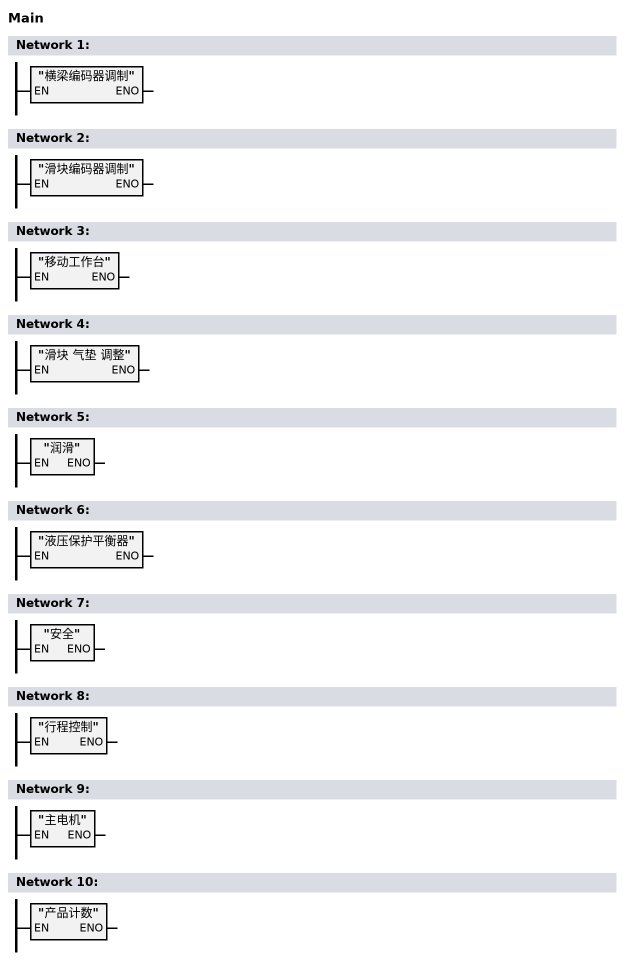
   RUNG wire#powerrail
      "横梁编码器调制"()
   END_RUNG
   // the same network as SCL:
   "横梁编码器调制"();
END_REGION

REGION Network 2
   RUNG wire#powerrail
      "滑块编码器调制"()
   END_RUNG
   // the same network as SCL:
   "滑块编码器调制"();
END_REGION

REGION Network 3
   RUNG wire#powerrail
      "移动工作台"()
   END_RUNG
   // the same network as SCL:
   "移动工作台"();
END_REGION

REGION Network 4
   RUNG wire#powerrail
      "滑块 气垫 调整"()
   END_RUNG
   // the same network as SCL:
   "滑块 气垫 调整"();
END_REGION

REGION Network 5
   RUNG wire#powerrail
      "润滑"()
   END_RUNG
   // the same network as SCL:
   "润滑"();
END_REGION

REGION Network 6
   RUNG wire#powerrail
      "液压保护平衡器"()
   END_RUNG
   // the same network as SCL:
   "液压保护平衡器"();
END_REGION

REGION Network 7
   RUNG wire#powerrail
      "安全"()
   END_RUNG
   // the same network as SCL:
   "安全"();
END_REGION

REGION Network 8
   RUNG wire#powerrail
      "行程控制"()
   END_RUNG
   // the same network as SCL:
   "行程控制"();
END_REGION

REGION Network 9
   RUNG wire#powerrail
      "主电机"()
   END_RUNG
   // the same network as SCL:
   "主电机"();
END_REGION

REGION Network 10
   RUNG wire#powerrail
      "产品计数"()
   END_RUNG
   // the same network as SCL:
   "产品计数"();
END_REGION
END_ORGANIZATION_BLOCK

(* ===== HMI "HMI_RT_1" =====
system functions are stored by id; their names below are inferred from use
connection "HMI_连接_1": ETHERNET, S7_1200_OMS

HMI tags "默认变量表"
   "360" : Bool = PLC 360 AT %M204.3, 100 ms
   "10度" : Bool = PLC 10度 AT %M200.0, 100 ms
   "20度" : Bool = PLC 20度 AT %M200.1, 100 ms
   "30度" : Bool = PLC 30度 AT %M200.2, 100 ms
   "40度" : Bool = PLC 40度 AT %M200.3, 100 ms
   "50" : Bool = PLC 50 AT %M200.4, 100 ms
   "60" : Bool = PLC 60 AT %M200.5, 100 ms
   "70" : Bool = PLC 70 AT %M200.6, 100 ms
   "80" : Bool = PLC 80 AT %M200.7, 100 ms
   "90" : Bool = PLC 90 AT %M201.0, 100 ms
   "100" : Bool = PLC 100 AT %M201.1, 100 ms
   "110" : Bool = PLC 110 AT %M201.2, 100 ms
   "120" : Bool = PLC 120 AT %M201.3, 100 ms
   "130" : Bool = PLC 130 AT %M201.4, 100 ms
   "140" : Bool = PLC 140 AT %M201.5, 100 ms
   "150" : Bool = PLC 150 AT %M201.6, 100 ms
   "160" : Bool = PLC 160 AT %M201.7, 100 ms
   "170" : Bool = PLC 170 AT %M202.0, 100 ms
   "180" : Bool = PLC 180 AT %M202.1, 100 ms
   "190" : Bool = PLC 190 AT %M202.2, 100 ms
   "200" : Bool = PLC 200 AT %M202.3, 100 ms
   "210" : Bool = PLC 210 AT %M202.4, 100 ms
   "220" : Bool = PLC 220 AT %M202.5, 100 ms
   "230" : Bool = PLC 230 AT %M202.6, 100 ms
   "240" : Bool = PLC 240 AT %M202.7, 100 ms
   "250" : Bool = PLC 250 AT %M203.0, 100 ms
   "260" : Bool = PLC 260 AT %M203.1, 100 ms
   "270" : Bool = PLC 270 AT %M203.2, 100 ms
   "280" : Bool = PLC 280 AT %M203.3, 100 ms
   "290" : Bool = PLC 290 AT %M203.4, 100 ms
   "300" : Bool = PLC 300 AT %M203.5, 100 ms
   "310" : Bool = PLC 310 AT %M203.6, 100 ms
   "320" : Bool = PLC 320 AT %M203.7, 100 ms
   "330" : Bool = PLC 330 AT %M204.0, 100 ms
   "340" : Bool = PLC 340 AT %M204.1, 100 ms
   "350" : Bool = PLC 350 AT %M204.2, 100 ms
   "工作台落到位前" : Bool = PLC "Tag_57(1)" AT %I7.3, 1 s
   "工作台落到位后" : Bool = PLC "Tag_58(1)" AT %I7.4, 1 s
   "工作台夹紧阀(1)" : Bool = PLC 左栅栏落下来检测 AT %Q13.1, 1 s
   "平衡缸气压检测" : Bool = PLC 平衡缸气压检测 AT %I10.5, 1 s
   "润滑油泵启动OK" : Bool = PLC 润滑油泵启动OK AT %M5.5, 1 s
   "润滑油压正常" : Bool = PLC 润滑油压正常 AT %M5.1, 1 s
   "液压保护故障" : Bool = PLC 液压保护故障 AT %M6.1, 1 s
   "横梁编码器" : DWord = PLC 横梁编码器 AT %ID68, 1 s
   "ECamdata _DB_+0.7" : DInt = PLC 滑块编码器 AT %ID72, 1 s
   "横梁编码器 _DB_+0.6" : Int = PLC "横梁编码器 _DB"."+0.6", 1 s
   "工作台放松阀(1)" : Bool = PLC "备用(16)" AT %Q13.2, 1 s
   "工作台落到位" : Bool = PLC 工作台落到位 AT %M7.1, 1 s
   "工作台-夹紧OK" : Bool = PLC "工作台-夹紧OK" AT %M15.2, 1 s
   "工作台放松OK" : Bool = PLC 工作台放松OK AT %M15.3, 1 s
   "横梁编码器 _DB_0.11" : Real = PLC "横梁编码器 _DB"."0.11", 1 s
   "滑块调整自动选择" : Bool = PLC 滑块调整自动选择 AT %M16.2, 1 s
   "ECamdata _DB_+0.36" : Int = PLC "ECamdata _DB"."+0.36", 100 ms
   "ECamdata _DB_+0.47" : Real = PLC "ECamdata _DB"."+0.47", 100 ms
   "ECamdata _DB_+0.6" : Int = PLC "ECamdata _DB".电子凸轮编码器显示, 100 ms
   "ECamdata _DB_AQD" : Real = PLC "ECamdata _DB".平衡器压力显示, 100 ms
   "ECamdata _DB_AQD2" : Real = PLC "ECamdata _DB".AQD2, 100 ms
   "ECamdata _DB_AQD3" : Real = PLC "ECamdata _DB".气垫模拟量显示1, 100 ms
   "ECamdata _DB_D{0}" : Real = PLC "ECamdata _DB".D[0], 100 ms
   "ECamdata _DB_D{1}" : Real = PLC "ECamdata _DB".D[1], 100 ms
   "ECamdata _DB_D{10}滑块设定高度" : Real = PLC "ECamdata _DB".D[10], 100 ms
   "ECamdata _DB_D{11}" : Real = PLC "ECamdata _DB".D[11], 100 ms
   "ECamdata _DB_D{6}" : Real = PLC "ECamdata _DB".D[6], 100 ms
   "ECamdata _DB_D{7}" : Real = PLC "ECamdata _DB".D[7], 100 ms
   "ECamdata _DB_D{9}" : Real = PLC "ECamdata _DB".D[9], 100 ms
   "ECamdata _DB_D102" : Int = PLC "ECamdata _DB".D102, 100 ms
   "ECamdata _DB_D107" : Int = PLC "ECamdata _DB".D107, 100 ms
   "ECamdata _DB_D108" : Real = PLC "ECamdata _DB".D108, 100 ms
   "ECamdata _DB_当前产量" : Int = PLC "ECamdata _DB".当前产量, 100 ms
   "ECamdata _DB_滑块打油次数" : Int = PLC "ECamdata _DB".滑块打油次数, 100 ms
   "ECamdata _DB_平衡器设置压力" : Real = PLC "ECamdata _DB".平衡器设置压力, 100 ms
   "ECamdata _DB_气垫2压力设置" : Real = PLC "ECamdata _DB".气垫2压力设置, 100 ms
   "ECamdata _DB_气垫模拟量显示1" : Real = PLC "ECamdata _DB".气垫模拟量显示2, 100 ms
   "ECamdata _DB_气垫压力设置" : Real = PLC "ECamdata _DB".气垫1压力设置, 100 ms
   "ECamdata _DB_设置产量" : Int = PLC "ECamdata _DB".设置产量, 100 ms
   "ECamdata _DB_主分油器打油次数" : Int = PLC "ECamdata _DB".主分油器打油次数, 100 ms
   "滑块调整手动/自动" : Bool = PLC "滑块调整手动/自动" AT %M301.5, 100 ms
   "ECamdata _DB_D{10}滑块设定高度(1)" : Real = PLC "ECamdata _DB_D{10}滑块设定高度" AT %MD150, 1 s
   "横梁编码器 _DB_+0.8" : Int = PLC "横梁编码器 _DB"."+0.8", 1 s
   "PLC报警变量组1" : Int = PLC PLC报警变量组1 AT %MW3000, 100 ms
   "PLC报警变量组2" : Int = PLC PLC报警变量组2 AT %MW3002, 1 s
   "上极限" : Bool = PLC 上极限 AT %I13.4, 1 s
   "工作台顶起" : Bool = PLC 工作台顶起 AT %Q11.4, 1 s
   "液压保护正常" : Bool = PLC 液压保护正常 AT %M207.6, 1 s
   "润滑正常" : Bool = PLC 润滑不正常 AT %M1000.4, 1 s
   "滑块调整电机空开" : Bool = PLC 滑块调整电机空开 AT %I2.1, 1 s
   "滑块调整选择开关" : Bool = PLC 滑块调整选择开关 AT %I10.0, 1 s
   "上死点" : Bool = PLC 上死点 AT %M204.4, 1 s
   "滑块调整上极限" : Bool = PLC 滑块调整上极限 AT %I10.3, 1 s
   "滑块调整下极限" : Bool = PLC 滑块调整下极限 AT %I10.4, 1 s
   "滑块调整向上" : Bool = PLC 滑块调整向上 AT %I10.1, 1 s
   "滑块调整向下" : Bool = PLC 滑块调整向下 AT %I10.2, 1 s
   "急停故障(2)" : Bool = PLC "急停故障(2)" AT %M300.0, 1 s
   "行程选择" : Bool = PLC 行程选择 AT %M207.3, 1 s
   "左后双手使用" : Bool = PLC 左后双手使用 AT %I4.4, 1 s
   "右前双手选择" : Bool = PLC 右前双手选择 AT %I25.2, 1 s
   "工作台放松顶起" : Bool = PLC 工作台放松顶起 AT %I14.4, 1 s
   "调整开关" : Bool = PLC 调整开关 AT %I14.5, 1 s
   "工作台顶起压力" : Bool = PLC 工作台顶起压力 AT %I15.3, 1 s
   "工作台顶起右前检测" : Bool = PLC 工作台顶起右前检测 AT %I17.3, 1 s
   "工作台顶起左后检测" : Bool = PLC 工作台顶起左后检测 AT %I17.4, 1 s
   "工作台落下右边后检测" : Bool = PLC 工作台落下右边后检测 AT %I18.1, 1 s
   "工作台落下右前检测" : Bool = PLC 工作台落下右前检测 AT %I17.7, 1 s
   "工作台落下左前检测" : Bool = PLC 工作台落下左前检测 AT %I17.6, 1 s
   "工作台落下左后检测" : Bool = PLC 工作台落下左后检测 AT %I18.0, 1 s
   "开工作台变频器正常" : Bool = PLC 开工作台变频器正常 AT %I2.6, 1 s
   "工作台开进" : Bool = PLC 工作台开进 AT %I15.0, 1 s
   "工作台开进到位" : Bool = PLC 工作台开进到位 AT %I16.2, 1 s
   "工作台开出" : Bool = PLC 工作台开出 AT %I14.7, 1 s
   "工作台左前顶起到位" : Bool = PLC 工作台左前顶起到位 AT %I15.6, 1 s
   "工作台右前顶起到位" : Bool = PLC 工作台右前顶起到位 AT %I15.7, 1 s
   "工作台左后顶起到位" : Bool = PLC 工作台左后顶起到位 AT %I16.0, 1 s
   "工作台右后顶起到位" : Bool = PLC 工作台右后顶起到位 AT %I16.1, 1 s
   "工作台落下夹紧(1)" : Bool = PLC "工作台落下夹紧(1)" AT %I14.3, 1 s
   "工作台放松顶起(1)" : Bool = PLC "工作台放松顶起(1)" AT %Q11.1, 1 s
   "工作台落下夹紧(2)" : Bool = PLC "工作台落下夹紧(2)" AT %Q11.3, 1 s
   "润滑电机工作指示" : Bool = PLC 润滑电机工作指示 AT %Q12.4, 1 s
   "正转条件" : Bool = PLC 正转条件 AT %M1000.7, 1 s
   "主电机启动指示" : Bool = PLC 主电机启动指示 AT %Q12.0, 1 s
   "主电机启动延时" : Bool = PLC 主电机启动延时 AT %M1100.4, 1 s
   "IEC_Counter_0_DB_4_CV" : Int = PLC 当前产量.CV, 100 ms
   "产量到达" : Bool = PLC 产量到达 AT %M30.2, 1 s
   "计数开始" : Bool = PLC 计数开始 AT %M30.0, 1 s
   "计数清零" : Bool = PLC 计数清零 AT %M30.1, 1 s
   "当前产量" : Time = PLC IEC_Timer_0_DB_4.PT, 1 s
   "IEC_Timer_0_DB_4" : Time = PLC IEC_Timer_0_DB_4.PT, 100 ms
   "主电机正转运行" : Bool = PLC 主电机正转运行 AT %Q2.0, 1 s
   "横梁1分油器检测" : Bool = PLC 横梁1分油器检测 AT %I5.1, 1 s
   "平衡器分油器检测" : Bool = PLC 平衡器分油器检测 AT %I5.0, 1 s
   "润滑故障" : Bool = PLC 润滑故障 AT %M15.4, 1 s
   "主电机零速" : Bool = PLC 主电机零速 AT %I2.5, 1 s
   "主电机温度检测(1)" : Bool = PLC "主电机温度检测(1)" AT %I4.1, 1 s
   "主电机调速装置正常" : Bool = PLC 主电机调速装置正常 AT %I2.4, 1 s
   "主电机风扇空开" : Bool = PLC 主电机风扇空开 AT %I2.3, 1 s
   "主电机风扇流量检测(1)" : Bool = PLC "主电机风扇流量检测(1)" AT %I4.0, 1 s
   "按钮站插入" : Bool = PLC 按钮站插入 AT %I15.5, 1 s
   "右前急停按钮" : Bool = PLC 右前急停按钮 AT %I22.4, 1 s
   "左前急停按钮" : Bool = PLC 左前急停按钮 AT %I22.5, 1 s
   "右后急停按钮" : Bool = PLC 右后急停按钮 AT %I22.6, 1 s
   "左后急停按钮" : Bool = PLC 左后急停按钮 AT %I22.7, 1 s
   "前安全栓" : Bool = PLC 前安全栓 AT %I23.1, 1 s
   "后安全栓" : Bool = PLC 后安全栓 AT %I23.0, 1 s
   "气垫调整空开" : Bool = PLC 气垫调整空开 AT %I2.2, 1 s
   "气垫调整上极限" : Bool = PLC 气垫调整上极限 AT %I11.2, 1 s
   "气垫调整下极限" : Bool = PLC 气垫调整下极限 AT %I11.3, 1 s
   "气垫冷却电机过热" : Bool = PLC 气垫冷却电机过热 AT %I13.1, 1 s
   "气垫左落下到位" : Bool = PLC 气垫左落下到位 AT %I11.6, 1 s
   "气垫压力检测" : Bool = PLC 气垫压力检测 AT %I12.1, 1 s
   "工作台顶起左前检测" : Bool = PLC 工作台顶起左前检测 AT %I17.2, 1 s
   "工作台顶起右后检测" : Bool = PLC 工作台顶起右后检测 AT %I17.5, 1 s
   "工作台左前落到为" : Bool = PLC 工作台左前落到为 AT %I16.3, 1 s
   "工作台右前落到为" : Bool = PLC 工作台右前落到为 AT %I16.4, 1 s
   "工作台左后落到为" : Bool = PLC 工作台左后落到为 AT %I16.5, 1 s
   "工作台右后落到位" : Bool = PLC 工作台右后落到位 AT %I16.6, 1 s
   "润滑电机空开" : Bool = PLC 润滑电机空开 AT %I3.0, 1 s
   "润滑油位检测" : Bool = PLC 润滑油位检测 AT %I21.1, 1 s
   "润滑过滤检测" : Bool = PLC 润滑过滤检测 AT %I21.2, 1 s
   "滑块分油器检测" : Bool = PLC 滑块分油器检测 AT %I22.1, 1 s
   "气垫分油器检测" : Bool = PLC 气垫分油器检测 AT %I22.2, 1 s
   "液压保护系统空开" : Bool = PLC 液压保护系统空开 AT %I2.7, 1 s
   "50/AR液压保护压力" : Bool = PLC "50/AR液压保护压力" AT %I18.6, 1 s
   "90/AR液压保护压力" : Bool = PLC "90/AR液压保护压力" AT %I18.7, 1 s
   "100/AR液压保护压力" : Bool = PLC "100/AR液压保护压力" AT %I18.4, 1 s
   "135/AR液压保护压力" : Bool = PLC "135/AR液压保护压力" AT %I18.5, 1 s
   "150/AR液压保护压力" : Bool = PLC "150/AR液压保护压力" AT %I19.0, 1 s
   "离制压力检测" : Bool = PLC 离制压力检测 AT %I24.0, 1 s
   "离制油箱油位检测" : Bool = PLC 离制油箱油位检测 AT %I24.2, 1 s
   "离制油箱油温检测" : Bool = PLC 离制油箱油温检测 AT %I24.6, 1 s
   "离制过滤器检测" : Bool = PLC 离制过滤器检测 AT %I23.7, 1 s
   "离制双阀反馈1" : Bool = PLC 离制双阀反馈1 AT %I3.4, 1 s
   "离制双阀反馈2" : Bool = PLC 离制双阀反馈2 AT %I3.5, 1 s
   "离合器油泵空开" : Bool = PLC 离合器油泵空开 AT %I3.6, 1 s
   "离合器运行" : Bool = PLC 离合器运行 AT %I3.7, 1 s
   "离合器准确检测" : Bool = PLC 离合器准确检测 AT %I5.2, 1 s
   "离合冷却过滤器检测" : Bool = PLC 离合冷却过滤器检测 AT %I24.3, 1 s
   "平衡缸进气阀" : Bool = PLC 平衡缸进气阀 AT %Q10.0, 1 s
   "平衡缸排气阀" : Bool = PLC 平衡缸排气阀 AT %Q10.1, 1 s
   "左气垫进气阀" : Bool = PLC 左气垫进气阀 AT %Q10.2, 1 s
   "左气垫排气阀" : Bool = PLC 左气垫排气阀 AT %Q10.3, 1 s
   "右气垫进气阀" : Bool = PLC 右气垫进气阀 AT %Q10.4, 1 s
   "右气垫气排阀" : Bool = PLC 右气垫气排阀 AT %Q10.5, 1 s
   "气动泵气源阀-1#" : Bool = PLC "气动泵气源阀-1#" AT %Q10.6, 1 s
   "液压保护泵启动（卸载）阀-2#" : Bool = PLC 气动泵气源阀 AT %Q10.7, 1 s
   "液压保护负荷荷 阀-3#" : Bool = PLC "液压保护负荷荷 阀-3#" AT %Q11.0, 1 s
   "平衡器间歇润滑阀" : Bool = PLC 平衡器间歇润滑阀 AT %Q0.2, 1 s
   "气垫间歇润滑阀" : Bool = PLC 气垫间歇润滑阀 AT %Q11.6, 1 s
   "自动化气压" : Bool = PLC 自动化气压 AT %Q11.7, 1 s
   "飞轮停止指示灯" : Bool = PLC 飞轮停止指示灯 AT %Q12.1, 1 s
   "模具移出指示" : Bool = PLC 模具移出指示 AT %Q12.2, 1 s
   "模具装入指示" : Bool = PLC 模具装入指示 AT %Q12.3, 1 s
   "液压保护正常指示" : Bool = PLC 液压保护故障 AT %M6.1, 1 s
   "液压保护卸荷指示" : Bool = PLC 液压保护卸荷指示 AT %Q12.6, 1 s
   "气垫升" : Bool = PLC 气垫升 AT %Q0.5, 1 s
   "气垫降" : Bool = PLC 气垫降 AT %Q0.6, 1 s
   "飞轮制动阀" : Bool = PLC 飞轮制动阀 AT %Q0.3, 1 s
   "单人操作" : Bool = PLC 单人操作 AT %Q0.4, 1 s
   "气垫升(1)" : Bool = PLC "气垫升(1)" AT %Q0.0, 1 s
   "气垫降(1)" : Bool = PLC "气垫降(1)" AT %Q0.1, 1 s
   "速度控制" : Bool = PLC 速度控制 AT %Q1.0, 1 s
   "主电机反转" : Bool = PLC 主电机反转 AT %Q1.1, 1 s
   "系统泵开始" : Bool = PLC 系统泵开始 AT %Q2.1, 1 s
   "变频器使能" : Bool = PLC 变频器使能 AT %Q2.2, 1 s
   "润滑电机" : Bool = PLC 润滑电机 AT %Q2.6, 1 s
   "工作台电机正转(1)" : Bool = PLC "工作台电机正转(1)" AT %Q2.3, 1 s
   "工作骀电机反转" : Bool = PLC 工作骀电机反转 AT %Q2.4, 1 s
   "工作台变速" : Bool = PLC 工作台变速 AT %Q2.5, 1 s
   "安全正常(1)" : Bool = PLC "安全正常(1)" AT %Q2.7, 1 s
   "压机急停1" : Bool = PLC 压机急停1 AT %Q3.0, 1 s
   "压机急停2" : Bool = PLC 压机急停2 AT %Q3.1, 1 s
   "离合器油泵电机" : Bool = PLC 离合器油泵电机 AT %Q3.2, 1 s
   "单次连续继电器" : Bool = PLC 单次连续继电器 AT %Q3.3, 1 s
   "滑块向上调整" : Bool = PLC 滑块向上调整 AT %Q3.4, 1 s
   "滑块向下调整" : Bool = PLC 滑块向下调整 AT %Q3.5, 1 s
   "主电机风扇运行" : Bool = PLC 主电机风扇运行 AT %Q3.6, 1 s
   "下死点" : Bool = PLC 下死点 AT %M204.6, 1 s
   "液压保护故障(1)" : Bool = PLC "液压保护故障(1)" AT %M208.0, 1 s

discrete alarms
   1: '急停', class Errors, trigger "PLC报警变量组1" bit 0
   2: '润滑压力异常', class Errors, trigger "PLC报警变量组1" bit 1
   3: '"离合器压力异常', class Errors, trigger "PLC报警变量组1" bit 2
   4: '"平衡器压力异常"', class Errors, trigger "PLC报警变量组1" bit 3
   5: '"液压保护过载"', class Errors, trigger "PLC报警变量组1" bit 4
   6: '"低液位"', class Errors, trigger "PLC报警变量组1" bit 5
   7: '"滑块调整上限位断开"', class Errors, trigger "PLC报警变量组1" bit 6
   8: '"滑块调整下限位断开"', class Errors, trigger "PLC报警变量组1" bit 7
   9: '"双阀粘连1-K3"', class Errors, trigger "PLC报警变量组1" bit 8
   10: '"双阀粘连1-K4"', class Errors, trigger "PLC报警变量组1" bit 9
   11: '"双阀继电器粘连1"', class Errors, trigger "PLC报警变量组1" bit 10
   12: '"双阀继电器粘连2"', class Errors, trigger "PLC报警变量组1" bit 11
   13: '"润滑电机过载"', class Errors, trigger "PLC报警变量组1" bit 12
   14: '"工作台油泵电机过载"', class Errors, trigger "PLC报警变量组1" bit 13
   15: '"主电机过载"', class Errors, trigger "PLC报警变量组1" bit 14
   16: '"润滑异常"', class Errors, trigger "PLC报警变量组1" bit 15
   17: '工作台未夹紧', class Errors, trigger "PLC报警变量组2" bit 0
   18: '"工作台未眠放松"', class Errors, trigger "PLC报警变量组2" bit 1
   19: '"液压保护压力未正常"', class Errors, trigger "PLC报警变量组2" bit 2
   20: '"滑块调整电机过载"', class Errors, trigger "PLC报警变量组2" bit 3
   21: '"超载指示"', class Errors, trigger "PLC报警变量组2" bit 4
   22: '"气压未正常"', class Errors, trigger "PLC报警变量组2" bit 5
   23: '"急停中', class Errors, trigger "PLC报警变量组2" bit 6
   24: '异常报警', class Errors, trigger "PLC报警变量组2" bit 7
   25: '右前工作台未落下到位', class Errors, trigger "PLC报警变量组2" bit 8
   26: '左后工作台未落下到位', class Errors, trigger "PLC报警变量组2" bit 9
   27: '"右前工作台未顶起到位"', class Errors, trigger "PLC报警变量组2" bit 10
   28: '"左前工作台未顶起到位"', class Errors, trigger "PLC报警变量组2" bit 11
   29: '"工作台未开进到位"', class Errors, trigger "PLC报警变量组2" bit 12
   30: '左气垫未落下到位', class Errors, trigger "PLC报警变量组2" bit 13
   31: '中气垫未落下到位', class Errors, trigger "PLC报警变量组2" bit 14
   32: '右气垫未落下到位', class Errors, trigger "PLC报警变量组2" bit 15

graphic list "@DiagnosticsStates": 0 '@Diagnostics_StateGood'; 1 '@Diagnostics_StateBad'

screen "滑块角度" 800x480
   Circle "圆_2" at 245,51 size 21x21
      Appearance <- "360"
   Circle "圆_3" at 274,56 size 21x21
      Appearance <- "10度"
   Circle "圆_4" at 303,66 size 21x21
      Appearance <- "20度"
   Circle "圆_5" at 326,79 size 21x21
      Appearance <- "30度"
   Circle "圆_6" at 346,95 size 21x21
      Appearance <- "40度"
   Circle "圆_7" at 364,115 size 21x21
      Appearance <- "50"
   Circle "圆_8" at 377,135 size 21x21
      Appearance <- "60"
   Circle "圆_9" at 385,157 size 21x21
      Appearance <- "70"
   Circle "圆_10" at 392,179 size 21x21
      Appearance <- "80"
   Circle "圆_11" at 394,202 size 21x21
      Appearance <- "90"
   Circle "圆_12" at 391,226 size 21x21
      Appearance <- "100"
   Circle "圆_13" at 386,249 size 21x21
      Appearance <- "110"
   Circle "圆_14" at 378,271 size 21x21
      Appearance <- "120"
   Circle "圆_15" at 365,292 size 21x21
      Appearance <- "130"
   Circle "圆_16" at 348,311 size 21x21
      Appearance <- "140"
   Circle "圆_17" at 328,328 size 21x21
      Appearance <- "150"
   Circle "圆_18" at 306,342 size 21x21
      Appearance <- "160"
   Circle "圆_19" at 276,353 size 21x21
      Appearance <- "170"
   Circle "圆_20" at 247,357 size 21x21
      Appearance <- "180"
   Circle "圆_22" at 219,352 size 21x21
      Appearance <- "190"
   Circle "圆_23" at 195,344 size 21x21
      Appearance <- "200"
   Circle "圆_24" at 172,333 size 21x21
      Appearance <- "210"
   Circle "圆_25" at 152,319 size 21x21
      Appearance <- "220"
   Circle "圆_26" at 133,302 size 21x21
      Appearance <- "230"
   Circle "圆_27" at 117,281 size 21x21
      Appearance <- "240"
   Circle "圆_28" at 104,258 size 21x21
      Appearance <- "250"
   Circle "圆_29" at 96,229 size 21x21
      Appearance <- "260"
   Circle "圆_30" at 93,201 size 21x21
      Appearance <- "270"
   Circle "圆_32" at 95,178 size 21x21
      Appearance <- "280"
   Circle "圆_33" at 100,155 size 21x21
      Appearance <- "290"
   Circle "圆_34" at 110,131 size 21x21
      Appearance <- "300"
   Circle "圆_35" at 126,111 size 21x21
      Appearance <- "310"
   Circle "圆_36" at 144,91 size 21x21
      Appearance <- "320"
   Circle "圆_37" at 167,74 size 21x21
      Appearance <- "330"
   Circle "圆_38" at 191,63 size 21x21
      Appearance <- "340"
   Circle "圆_39" at 218,54 size 21x21
      Appearance <- "350"
   TextField "文本域_2" at 422,193 size 43x40; Text '90'
   TextField "文本域_3" at 221,378 size 62x40; Text '180'
   TextField "文本域_5" at 196,174 size 117x31; Text '滑块位置'
   TextField "文本域_9" at 467,193 size 93x25; Text '当前产量'
   TextField "文本域_4" at 25,203 size 62x40; Text '270'
   TextField "文本域_1" at 241,12 size 24x40; Text '0'
   SymbolLibrary "符号库_1" at 405,7 size 109x71
   SymbolLibrary "符号库_2" at 646,29 size 86x40
   TextField "文本域_7" at 637,83 size 77x21; Text '滑块电机'
   TextField "文本域_6" at 423,85 size 59x21; Text '主电机'
   TextField "文本域_8" at 467,127 size 93x25; Text '设置产量'
   TextField "文本域_10" at 693,127 size 93x25; Text '计数清零'
   TextField "文本域_13" at 586,126 size 93x25; Text '计数通断'
   TextField "文本域_11" at 19,335 size 93x25; Text '润滑检测'
   TextField "文本域_15" at 583,14 size 33x17; Text '向上'
   TextField "文本域_16" at 738,15 size 33x17; Text '向下'
   Button "按钮_1" at 28,424 size 67x56; TextOff '滑块角度'
      on Click: ActivateScreen("滑块角度", 0)
   Button "按钮_2" at 96,424 size 67x56; TextOff '设备状态'
      on Click: ActivateScreen("设备状态", 0)
   Button "按钮_3" at 163,424 size 71x55; TextOff '工作台操作'
      on Click: ActivateScreen("工作台操作", 0)
   Button "按钮_4" at 235,424 size 69x56; TextOff '气垫操作'
      on Click: ActivateScreen("气垫操作", 0)
   Button "按钮_5" at 304,423 size 66x57; TextOff '故障显示'
      on Click: ActivateScreen("故障显示", 0)
   Button "按钮_6" at 371,423 size 73x57; TextOff '输出显示'
      on Click: ActivateScreen("输出显示", 0)
   Button "按钮_7" at 445,422 size 66x58; TextOff '输入显示'
      on Click: ActivateScreen("输入显示", 0)
   IOField "I/O 域_1" at 228,215 size 56x32; FormatPattern 999
      ProcessValue <- "横梁编码器 _DB_+0.6"
   IOField "I/O 域_2" at 478,153 size 81x29; FormatPattern 9999
      ProcessValue <- "ECamdata _DB_设置产量"
   Button "按钮_8" at 514,423 size 68x56; TextOn '滑块调整'; TextOff '滑块调整'
      on Click: ActivateScreen("滑块调整", 0)
   Button "按钮_9" at 667,421 size 65x58; TextOff '报警信息'
      on Click: ActivateScreen("报警信息", 0)
   Button "按钮_10" at 585,423 size 77x55; TextOff '行程控制'
      on Click: ActivateScreen("行程控制", 0)
   Circle "圆_1" at 436,26 size 35x35
      Appearance <- "主电机正转运行"
   Circle "圆_21" at 584,33 size 33x33
      Appearance <- "滑块调整向上"
   Circle "圆_31" at 738,34 size 33x33
      Appearance <- "滑块调整向下"
   IOField "I/O 域_3" at 478,219 size 87x32; FormatPattern 9999
      ProcessValue <- "IEC_Counter_0_DB_4_CV"
   Rectangle "矩形_1" at 479,258 size 88x60
      Appearance <- "产量到达"
   TextField "文本域_14" at 478,277 size 85x23; Text '产量完成'
   Switch "开关_1" at 579,170 size 102x93; CaptionText 'Switch'; TextOff '断'; TextOn '通'
      ProcessValue <- "计数开始"
      Appearance <- "计数开始"
   Button "按钮_11" at 702,187 size 75x72; TextOff '清零'
      on Press: function_b14e0dd5("计数清零", 0)
   Circle "圆_42" at 25,371 size 35x35
      Appearance <- "横梁1分油器检测"
   Circle "圆_43" at 72,372 size 35x35
      Appearance <- "平衡器分油器检测"
   Circle "圆_45" at 227,101 size 55x55
      Appearance <- "上死点"
   Circle "圆_46" at 226,275 size 55x55
      Appearance <- "下死点"
   TextField "文本域_12" at 383,338 size 93x25; Text '润滑故障'
   Circle "圆_44" at 423,372 size 35x35
      Appearance <- "润滑正常"
   TextField "文本域_19" at 593,338 size 93x25; Text '平衡气压'
   Circle "圆_47" at 633,373 size 35x35
      Appearance <- "平衡缸气压检测"
   TextField "文本域_20" at 690,338 size 93x25; Text '液压保护'
   Circle "圆_48" at 730,372 size 35x35
      Appearance <- "液压保护正常"
   TextField "文本域_21" at 491,339 size 93x25; Text '离制压力'
   Circle "圆_49" at 529,371 size 35x35
      Appearance <- "离制压力检测"

screen "设备状态" 800x480
   TextField "文本域_1" at 63,79 size 101x27; Text '润滑正常'
   TextField "文本域_2" at 64,142 size 101x27; Text '急停正常'
   TextField "文本域_3" at 50,205 size 125x27; Text '工作台夹紧'
   TextField "文本域_4" at 66,268 size 101x27; Text '气压正常'
   TextField "文本域_5" at 46,331 size 149x27; Text '液压保护正常'
   Circle "圆_1" at 325,208 size 27x27
      Appearance <- "工作台落到位前"
   TextField "文本域_6" at 293,237 size 96x16; Text '工作台前落到为'
   Circle "圆_2" at 427,207 size 27x27
      Appearance <- "工作台落到位后"
   TextField "文本域_7" at 395,237 size 96x16; Text '工作台后落到为'
   TextField "文本域_8" at 495,237 size 96x16; Text '工作台夹紧压力'
   Circle "圆_4" at 223,207 size 27x27
      Appearance <- "工作台夹紧阀(1)"
   TextField "文本域_9" at 198,237 size 83x16; Text '工作台夹紧阀'
   Circle "圆_5" at 427,81 size 27x27
      Appearance <- "润滑油压正常"
   TextField "文本域_10" at 399,111 size 83x16; Text '润滑油压正常'
   TextField "文本域_12" at 295,111 size 96x16; Text '润滑过滤器正常'
   Circle "圆_8" at 222,81 size 27x27
      Appearance <- "工作台落到位后"
   TextField "文本域_13" at 196,111 size 83x16; Text '润滑油位正常'
   Circle "圆_9" at 527,81 size 27x27
      Appearance <- "工作台落到位后"
   TextField "文本域_14" at 502,111 size 83x16; Text '润滑频次正常'
   Circle "圆_10" at 325,270 size 27x27
      Appearance <- "工作台落到位前"
   TextField "文本域_15" at 306,299 size 70x16; Text '离合器压力'
   Circle "圆_11" at 427,269 size 27x27
      Appearance <- "工作台落到位后"
   Circle "圆_12" at 223,269 size 27x27
      Appearance <- "平衡缸气压检测"
   TextField "文本域_16" at 200,298 size 70x16; Text '平衡缸压力'
   TextField "文本域_17" at 407,300 size 70x16; Text '制动器压力'
   Circle "圆_6" at 615,81 size 27x27
      Appearance <- "润滑油泵启动OK"
   TextField "文本域_11" at 590,111 size 83x16; Text '润滑电机启动'
   TextField "文本域_19" at 312,171 size 57x16; Text '急停闭点'
   TextField "文本域_20" at 207,171 size 57x16; Text '急停开点'
   TextField "文本域_21" at 414,171 size 57x16; Text '梯子开关'
   TextField "文本域_23" at 306,362 size 70x16; Text '卸荷阀卸荷'
   Circle "圆_19" at 427,332 size 27x27
      Appearance <- "液压保护故障"
   TextField "文本域_24" at 200,361 size 83x16; Text '液压保护压力'
   TextField "文本域_25" at 407,363 size 57x16; Text '系统压力'
   Button "按钮_1" at 28,424 size 67x56; TextOn '滑块角度'; TextOff '滑块角度'
      on Click: ActivateScreen("滑块角度", 0)
   Button "按钮_2" at 96,424 size 67x56; TextOn '设备状态'; TextOff '设备状态'
      on Click: ActivateScreen("设备状态", 0)
   Button "按钮_3" at 163,424 size 71x55; TextOn '工作台操作'; TextOff '工作台操作'
      on Click: ActivateScreen("工作台操作", 0)
   Button "按钮_4" at 235,424 size 69x56; TextOn '气垫操作'; TextOff '气垫操作'
      on Click: ActivateScreen("气垫操作", 0)
   Button "按钮_5" at 304,423 size 66x57; TextOn '故障显示'; TextOff '故障显示'
      on Click: ActivateScreen("故障显示", 0)
   Button "按钮_6" at 371,423 size 73x57; TextOn '输出显示'; TextOff '输出显示'
      on Click: ActivateScreen("输出显示", 0)
   Button "按钮_7" at 445,422 size 66x58; TextOn '输入显示'; TextOff '输入显示'
      on Click: ActivateScreen("输入显示", 0)
   Button "按钮_8" at 514,423 size 68x56; TextOn '滑块调整'; TextOff '滑块调整'
      on Click: ActivateScreen("滑块调整", 0)
   Button "按钮_9" at 592,422 size 65x58; TextOn '报警信息'; TextOff '报警信息'
      on Click: ActivateScreen("报警信息", 0)

screen "输入显示" 800x480
   Button "按钮_1" at 28,424 size 67x56; TextOn '滑块角度'; TextOff '滑块角度'
      on Click: ActivateScreen("滑块角度", 0)
   Button "按钮_2" at 96,424 size 67x56; TextOn '设备状态'; TextOff '设备状态'
      on Click: ActivateScreen("设备状态", 0)
   Button "按钮_3" at 163,424 size 71x55; TextOn '工作台操作'; TextOff '工作台操作'
      on Click: ActivateScreen("工作台操作", 0)
   Button "按钮_4" at 235,424 size 69x56; TextOn '气垫操作'; TextOff '气垫操作'
      on Click: ActivateScreen("气垫操作", 0)
   Button "按钮_5" at 304,423 size 66x57; TextOn '故障显示'; TextOff '故障显示'
      on Click: ActivateScreen("故障显示", 0)
   Button "按钮_6" at 371,423 size 73x57; TextOn '输出显示'; TextOff '输出显示'
      on Click: ActivateScreen("输出显示", 0)
   Button "按钮_7" at 445,422 size 66x58; TextOn '输入显示'; TextOff '输入显示'
      on Click: ActivateScreen("输入显示", 0)
   Button "按钮_8" at 514,423 size 68x56; TextOn '滑块调整'; TextOff '滑块调整'
      on Click: ActivateScreen("滑块调整", 0)
   Button "按钮_9" at 592,422 size 65x58; TextOn '报警信息'; TextOff '报警信息'
      on Click: ActivateScreen("报警信息", 0)
   TextField "文本域_1" at 10,10 size 112x19; Text '主电机零速'
      Appearance <- "主电机零速"
   TextField "文本域_2" at 10,40 size 117x19; Text '主电机温度检测'
      Appearance <- "主电机温度检测(1)"
   TextField "文本域_3" at 10,70 size 117x19; Text '调速装置正常'
      Appearance <- "主电机调速装置正常"
   TextField "文本域_4" at 10,100 size 117x19; Text '主电机风扇空开'
      Appearance <- "主电机风扇空开"
   TextField "文本域_5" at 10,130 size 117x19; Text '风扇流量检测'
      Appearance <- "主电机风扇流量检测(1)"
   TextField "文本域_8" at 10,220 size 112x19; Text '按钮站插入'
      Appearance <- "按钮站插入"
   TextField "文本域_9" at 10,250 size 112x19; Text '右前急停按钮'
      Appearance <- "右前急停按钮"
   TextField "文本域_10" at 10,280 size 112x19; Text '左前急停按钮'
      Appearance <- "左前急停按钮"
   TextField "文本域_11" at 10,310 size 112x19; Text '右后急停按钮'
      Appearance <- "右后急停按钮"
   TextField "文本域_12" at 10,340 size 112x19; Text '左后急停按钮'
      Appearance <- "左后急停按钮"
   TextField "文本域_13" at 10,370 size 112x19; Text '前安全栓'
      Appearance <- "前安全栓"
   TextField "文本域_14" at 10,400 size 112x19; Text '后安全栓'
      Appearance <- "后安全栓"
   TextField "文本域_15" at 150,220 size 119x19; Text '气垫调整空开'
      Appearance <- "气垫调整空开"
   TextField "文本域_16" at 150,250 size 119x19; Text '气垫调整上极限'
      Appearance <- "气垫调整上极限"
   TextField "文本域_17" at 150,280 size 119x19; Text '气垫调整上极限'
      Appearance <- "气垫调整下极限"
   TextField "文本域_18" at 150,310 size 119x19; Text '冷却电机过热'
      Appearance <- "气垫冷却电机过热"
   TextField "文本域_19" at 150,340 size 119x19; Text '气垫左落下到位'
      Appearance <- "气垫左落下到位"
   TextField "文本域_20" at 150,370 size 119x19; Text '气垫左落下到位'
      Appearance <- "气垫左落下到位"
   TextField "文本域_21" at 150,400 size 119x19; Text '气垫压力检测'
      Appearance <- "气垫压力检测"
   TextField "文本域_22" at 290,220 size 117x19; Text '工作台开进到位'
      Appearance <- "工作台开进到位"
   TextField "文本域_23" at 290,250 size 117x19; Text '左前落到为'
      Appearance <- "工作台左前落到为"
   TextField "文本域_24" at 290,280 size 117x19; Text '右前落到为'
      Appearance <- "工作台右前落到为"
   TextField "文本域_25" at 290,310 size 117x19; Text '左后落到为'
      Appearance <- "工作台左后落到为"
   TextField "文本域_26" at 290,340 size 117x19; Text '右后落到位'
      Appearance <- "工作台右后落到位"
   TextField "文本域_27" at 290,370 size 117x19; Text '工作台落下夹紧'
      Appearance <- "工作台落下夹紧(1)"
   TextField "文本域_29" at 430,220 size 114x19; Text '液保空开'
      Appearance <- "液压保护系统空开"
   TextField "文本域_30" at 430,250 size 114x19; Text '50/AR液保压力'
      Appearance <- "50/AR液压保护压力"
   TextField "文本域_31" at 430,280 size 114x19; Text '90/AR液保压力'
      Appearance <- "90/AR液压保护压力"
   TextField "文本域_32" at 430,310 size 123x19; Text '100/AR液保压力'
      Appearance <- "100/AR液压保护压力"
   TextField "文本域_33" at 430,340 size 123x19; Text '135/AR液保压力'
      Appearance <- "135/AR液压保护压力"
   TextField "文本域_34" at 430,370 size 123x19; Text '150/AR液保压力'
      Appearance <- "150/AR液压保护压力"
   TextField "文本域_35" at 430,400 size 117x19; Text '平衡缸气压检测'
      Appearance <- "平衡缸气压检测"
   TextField "文本域_37" at 570,250 size 117x19; Text '离合器运行'
      Appearance <- "离合器运行"
   TextField "文本域_38" at 570,280 size 117x19; Text '离合器准确检测'
      Appearance <- "离合器准确检测"
   TextField "文本域_39" at 570,310 size 117x19; Text '离合冷却过滤器'
      Appearance <- "离合冷却过滤器检测"
   TextField "文本域_43" at 150,10 size 119x19; Text '滑块调整空开'
      Appearance <- "滑块调整电机空开"
   TextField "文本域_44" at 150,40 size 119x19; Text '滑块调整选择'
      Appearance <- "滑块调整选择开关"
   TextField "文本域_45" at 150,70 size 119x19; Text '滑块调整向上'
      Appearance <- "滑块调整向上"
   TextField "文本域_46" at 150,100 size 119x19; Text '滑块调整向下'
      Appearance <- "滑块调整向下"
   TextField "文本域_47" at 150,130 size 119x19; Text '滑块调整上极限'
      Appearance <- "滑块调整上极限"
   TextField "文本域_48" at 150,160 size 119x19; Text '滑块调整下极限'
      Appearance <- "滑块调整下极限"
   TextField "文本域_50" at 290,10 size 115x19; Text '工作台顶起压力'
      Appearance <- "工作台顶起压力"
   TextField "文本域_51" at 290,40 size 115x19; Text '左前顶起到位'
      Appearance <- "工作台左前顶起到位"
   TextField "文本域_52" at 290,70 size 115x19; Text '右前顶起到位'
      Appearance <- "工作台右前顶起到位"
   TextField "文本域_53" at 290,100 size 115x19; Text '左后顶起到位'
      Appearance <- "工作台左后顶起到位"
   TextField "文本域_54" at 290,130 size 115x19; Text '右后顶起到位'
      Appearance <- "工作台右后顶起到位"
   TextField "文本域_57" at 430,10 size 101x19; Text '润滑电机空开'
      Appearance <- "润滑电机空开"
   TextField "文本域_58" at 430,40 size 101x19; Text '润滑油位检测'
      Appearance <- "润滑油位检测"
   TextField "文本域_59" at 430,70 size 101x19; Text '润滑过滤检测'
      Appearance <- "润滑过滤检测"
   TextField "文本域_60" at 430,100 size 101x19; Text '滑块分油器'
      Appearance <- "滑块分油器检测"
   TextField "文本域_61" at 430,130 size 101x19; Text '平衡器分油器'
      Appearance <- "平衡器分油器检测"
   TextField "文本域_62" at 430,160 size 101x19; Text '气垫分油器'
      Appearance <- "气垫分油器检测"
   TextField "文本域_63" at 430,190 size 101x19; Text '横梁1分油器'
      Appearance <- "横梁1分油器检测"
   TextField "文本域_64" at 570,10 size 117x19; Text '离制压力检测'
      Appearance <- "离制压力检测"
   TextField "文本域_65" at 570,40 size 117x19; Text '离制油位检测'
      Appearance <- "离制油箱油位检测"
   TextField "文本域_66" at 570,70 size 117x19; Text '离制油温检测'
      Appearance <- "离制油箱油温检测"
   TextField "文本域_67" at 570,100 size 117x19; Text '离制过滤器检测'
      Appearance <- "离制过滤器检测"
   TextField "文本域_68" at 570,130 size 117x19; Text '离制双阀反馈1'
      Appearance <- "离制双阀反馈1"
   TextField "文本域_69" at 570,160 size 117x19; Text '离制双阀反馈2'
      Appearance <- "离制双阀反馈2"
   TextField "文本域_70" at 569,220 size 117x19; Text '离合器油泵空开'
      Appearance <- "离合器油泵空开"
   TextField "文本域_6" at 290,160 size 115x19; Text '变频器正常'
      Appearance <- "开工作台变频器正常"

screen "输出显示" 800x480
   Button "按钮_1" at 28,424 size 67x56; TextOn '滑块角度'; TextOff '滑块角度'
      on Click: ActivateScreen("滑块角度", 0)
   Button "按钮_2" at 96,424 size 67x56; TextOn '设备状态'; TextOff '设备状态'
      on Click: ActivateScreen("设备状态", 0)
   Button "按钮_3" at 163,424 size 71x55; TextOn '工作台操作'; TextOff '工作台操作'
      on Click: ActivateScreen("工作台操作", 0)
   Button "按钮_4" at 235,424 size 69x56; TextOn '气垫操作'; TextOff '气垫操作'
      on Click: ActivateScreen("气垫操作", 0)
   Button "按钮_5" at 304,423 size 66x57; TextOn '故障显示'; TextOff '故障显示'
      on Click: ActivateScreen("故障显示", 0)
   Button "按钮_6" at 371,423 size 73x57; TextOn '输出显示'; TextOff '输出显示'
      on Click: ActivateScreen("输出显示", 0)
   Button "按钮_7" at 445,422 size 66x58; TextOn '输入显示'; TextOff '输入显示'
      on Click: ActivateScreen("输入显示", 0)
   Button "按钮_8" at 514,423 size 68x56; TextOn '滑块调整'; TextOff '滑块调整'
      on Click: ActivateScreen("滑块调整", 0)
   Button "按钮_9" at 592,422 size 65x58; TextOn '报警信息'; TextOff '报警信息'
      on Click: ActivateScreen("报警信息", 0)
   TextField "文本域_1" at 10,10 size 101x19; Text '平衡缸进气阀'
      Appearance <- "平衡缸进气阀"
   TextField "文本域_2" at 10,40 size 101x19; Text '平衡缸排气阀'
      Appearance <- "平衡缸排气阀"
   TextField "文本域_3" at 10,70 size 101x19; Text '左气垫进气阀'
      Appearance <- "左气垫进气阀"
   TextField "文本域_4" at 10,100 size 101x19; Text '左气垫排气阀'
      Appearance <- "左气垫排气阀"
   TextField "文本域_5" at 10,130 size 101x19; Text '右气垫进气阀'
      Appearance <- "右气垫进气阀"
   TextField "文本域_6" at 11,156 size 101x19; Text '右气垫排气阀'
      Appearance <- "右气垫气排阀"
   TextField "文本域_7" at 12,218 size 101x19; Text '气动泵气源阀'
      Appearance <- "气动泵气源阀-1#"
   TextField "文本域_8" at 12,248 size 117x19; Text '液保启动卸荷阀'
      Appearance <- "液压保护泵启动（卸载）阀-2#"
   TextField "文本域_9" at 12,278 size 85x19; Text '液保负荷阀'
      Appearance <- "液压保护负荷荷 阀-3#"
   TextField "文本域_10" at 12,308 size 117x19; Text '工作台放松顶起'
      Appearance <- "工作台放松顶起(1)"
   TextField "文本域_11" at 12,338 size 117x19; Text '工作台落下夹紧'
      Appearance <- "工作台落下夹紧(1)"
   TextField "文本域_12" at 13,364 size 101x19; Text '外工作台顶起'
      Appearance <- "工作台顶起"
   TextField "文本域_13" at 14,391 size 101x19; Text '外工作台落下'
      Appearance <- "工作台落下夹紧(2)"
   TextField "文本域_14" at 152,10 size 117x19; Text '气垫间歇润滑阀'
      Appearance <- "气垫间歇润滑阀"
   TextField "文本域_15" at 152,40 size 85x19; Text '自动化气压'
      Appearance <- "自动化气压"
   TextField "文本域_16" at 152,70 size 117x19; Text '主电机启动指示'
      Appearance <- "主电机启动指示"
   TextField "文本域_17" at 152,100 size 101x19; Text '飞轮停止指示'
      Appearance <- "飞轮停止指示灯"
   TextField "文本域_18" at 152,130 size 101x19; Text '模具移出指示'
      Appearance <- "模具移出指示"
   TextField "文本域_19" at 153,156 size 101x19; Text '模具装入指示'
      Appearance <- "模具装入指示"
   TextField "文本域_20" at 149,183 size 133x19; Text '润滑电机工作指示'
      Appearance <- "润滑电机工作指示"
   TextField "文本域_21" at 10,183 size 133x19; Text '平衡缸间歇润滑阀'
      Appearance <- "平衡器间歇润滑阀"
   TextField "文本域_22" at 157,219 size 133x19; Text '液压保护正常指示'
      Appearance <- "液压保护正常指示"
   TextField "文本域_23" at 157,249 size 133x19; Text '液压保护卸荷指示'
      Appearance <- "液压保护卸荷指示"
   TextField "文本域_24" at 157,279 size 85x19; Text '气垫升指示'
      Appearance <- "气垫升"
   TextField "文本域_25" at 157,309 size 85x19; Text '气垫降指示'
      Appearance <- "气垫降"
   TextField "文本域_26" at 157,339 size 85x19; Text '飞轮制动阀'
      Appearance <- "飞轮制动阀"
   TextField "文本域_27" at 158,365 size 69x19; Text '单人操作'
      Appearance <- "单人操作"
   TextField "文本域_28" at 154,392 size 85x19; Text '气垫电机升'
      Appearance <- "气垫升(1)"
   TextField "文本域_29" at 297,12 size 85x19; Text '气垫电机降'
      Appearance <- "气垫降(1)"
   TextField "文本域_30" at 297,42 size 85x19; Text '主电机运行'
      Appearance <- "主电机正转运行"
   TextField "文本域_31" at 297,72 size 69x19; Text '速度控制'
      Appearance <- "速度控制"
   TextField "文本域_32" at 297,102 size 85x19; Text '主电机反转'
      Appearance <- "主电机反转"
   TextField "文本域_33" at 297,132 size 85x19; Text '主电机正转'
      Appearance <- "主电机正转运行"
   TextField "文本域_34" at 298,158 size 85x19; Text '系统泵开始'
      Appearance <- "系统泵开始"
   TextField "文本域_35" at 294,185 size 101x19; Text '工台变频使能'
      Appearance <- "变频器使能"
   TextField "文本域_36" at 299,222 size 101x19; Text '工台电机正转'
      Appearance <- "工作台电机正转(1)"
   TextField "文本域_37" at 299,252 size 101x19; Text '工台电机反转'
      Appearance <- "工作骀电机反转"
   TextField "文本域_38" at 299,282 size 85x19; Text '工作台变速'
      Appearance <- "工作台变速"
   TextField "文本域_39" at 299,312 size 101x19; Text '润滑电机运行'
      Appearance <- "润滑电机"
   TextField "文本域_40" at 299,342 size 69x19; Text '安全正常'
      Appearance <- "安全正常(1)"
   TextField "文本域_41" at 300,368 size 78x19; Text '压机急停1'
      Appearance <- "压机急停1"
   TextField "文本域_42" at 296,395 size 78x19; Text '压机急停2'
      Appearance <- "压机急停2"
   TextField "文本域_43" at 439,13 size 117x19; Text '离合器油泵电机'
      Appearance <- "离合器油泵电机"
   TextField "文本域_44" at 439,43 size 117x19; Text '单次连续继电器'
      Appearance <- "单次连续继电器"
   TextField "文本域_45" at 439,73 size 101x19; Text '滑块向上调整'
      Appearance <- "滑块向上调整"
   TextField "文本域_46" at 439,103 size 101x19; Text '滑块向下调整'
      Appearance <- "滑块向下调整"
   TextField "文本域_47" at 439,133 size 117x19; Text '主电机风扇运行'
      Appearance <- "主电机风扇运行"

screen "故障显示" 800x480
   Button "按钮_1" at 28,424 size 67x56; TextOn '滑块角度'; TextOff '滑块角度'
      on Click: ActivateScreen("滑块角度", 0)
   Button "按钮_2" at 96,424 size 67x56; TextOn '设备状态'; TextOff '设备状态'
      on Click: ActivateScreen("设备状态", 0)
   Button "按钮_3" at 163,424 size 71x55; TextOn '工作台操作'; TextOff '工作台操作'
      on Click: ActivateScreen("工作台操作", 0)
   Button "按钮_4" at 235,424 size 69x56; TextOn '气垫操作'; TextOff '气垫操作'
      on Click: ActivateScreen("气垫操作", 0)
   Button "按钮_5" at 304,423 size 66x57; TextOn '故障显示'; TextOff '故障显示'
      on Click: ActivateScreen("故障显示", 0)
   Button "按钮_6" at 371,423 size 73x57; TextOn '输出显示'; TextOff '输出显示'
      on Click: ActivateScreen("输出显示", 0)
   Button "按钮_7" at 445,422 size 66x58; TextOn '输入显示'; TextOff '输入显示'
      on Click: ActivateScreen("输入显示", 0)
   Button "按钮_8" at 514,423 size 68x56; TextOn '滑块调整'; TextOff '滑块调整'
      on Click: ActivateScreen("滑块调整", 0)
   Button "按钮_9" at 592,422 size 65x58; TextOn '报警信息'; TextOff '报警信息'
      on Click: ActivateScreen("报警信息", 0)

screen "工作台操作" 800x480
   Button "按钮_1" at 28,424 size 67x56; TextOn '滑块角度'; TextOff '滑块角度'
      on Click: ActivateScreen("滑块角度", 0)
   Button "按钮_2" at 96,424 size 67x56; TextOn '设备状态'; TextOff '设备状态'
      on Click: ActivateScreen("设备状态", 0)
   Button "按钮_3" at 163,424 size 71x55; TextOn '工作台操作'; TextOff '工作台操作'
      on Click: ActivateScreen("工作台操作", 0)
   Button "按钮_4" at 235,424 size 69x56; TextOn '气垫操作'; TextOff '气垫操作'
      on Click: ActivateScreen("气垫操作", 0)
   Button "按钮_5" at 304,423 size 66x57; TextOn '故障显示'; TextOff '故障显示'
      on Click: ActivateScreen("故障显示", 0)
   Button "按钮_6" at 371,423 size 73x57; TextOn '输出显示'; TextOff '输出显示'
      on Click: ActivateScreen("输出显示", 0)
   Button "按钮_7" at 445,422 size 66x58; TextOn '输入显示'; TextOff '输入显示'
      on Click: ActivateScreen("输入显示", 0)
   TextField "文本域_1" at 47,68 size 125x27; Text '工作台松开'
   TextField "文本域_2" at 53,142 size 125x27; Text '工作台夹紧'
   Circle "圆_7" at 315,60 size 27x27
      Appearance <- "工作台放松顶起"
   TextField "文本域_12" at 308,92 size 44x16; Text '工作台'
   Circle "圆_8" at 222,60 size 27x27
      Appearance <- "上死点"
   TextField "文本域_13" at 215,92 size 44x16; Text '上死点'
   TextField "文本域_14" at 576,92 size 44x16; Text '工作台'
   Circle "圆_6" at 635,60 size 27x27
      Appearance <- "工作台放松OK"
   TextField "文本域_11" at 628,92 size 44x16; Text '工作台'
   Button "按钮_8" at 514,423 size 68x56; TextOn '滑块调整'; TextOff '滑块调整'
      on Click: ActivateScreen("滑块调整", 0)
   Button "按钮_9" at 592,422 size 65x58; TextOn '报警信息'; TextOff '报警信息'
      on Click: ActivateScreen("报警信息", 0)
   Circle "圆_1" at 271,60 size 27x27
      Appearance <- "调整开关"
   TextField "文本域_5" at 268,93 size 31x16; Text '调整'
   Circle "圆_3" at 582,60 size 27x27
      Appearance <- "工作台顶起压力"
   TextField "文本域_6" at 267,110 size 33x17; Text '开关'
   TextField "文本域_7" at 312,109 size 33x17; Text '顶起'
   TextField "文本域_8" at 574,110 size 47x17; Text '松压力'
   TextField "文本域_10" at 397,91 size 31x16; Text '前左'
   Circle "圆_4" at 399,60 size 27x27
      Appearance <- "工作台左前顶起到位"
   TextField "文本域_15" at 392,108 size 47x17; Text '松到位'
   TextField "文本域_16" at 443,91 size 31x16; Text '前右'
   Circle "圆_5" at 443,60 size 27x27
      Appearance <- "工作台右前顶起到位"
   TextField "文本域_17" at 438,109 size 47x17; Text '松到位'
   TextField "文本域_18" at 488,91 size 31x16; Text '后左'
   Circle "圆_9" at 489,60 size 27x27
      Appearance <- "工作台左后顶起到位"
   TextField "文本域_22" at 484,109 size 47x17; Text '松到位'
   TextField "文本域_23" at 535,91 size 31x16; Text '后右'
   Circle "圆_10" at 535,60 size 27x27
      Appearance <- "工作台右后顶起到位"
   TextField "文本域_24" at 530,109 size 47x17; Text '松到位'
   TextField "文本域_9" at 628,109 size 45x16; Text '松开OK'
   TextField "文本域_3" at 351,92 size 44x16; Text '工作台'
   Circle "圆_2" at 358,60 size 27x27
      Appearance <- "工作台放松顶起(1)"
   TextField "文本域_4" at 349,108 size 47x17; Text '松开阀'
   Circle "圆_11" at 268,141 size 27x27
      Appearance <- "工作台落下夹紧(1)"
   TextField "文本域_19" at 261,171 size 44x16; Text '工作台'
   TextField "文本域_21" at 529,170 size 44x16; Text '工作台'
   Circle "圆_13" at 588,141 size 27x27
      Appearance <- "工作台-夹紧OK"
   TextField "文本域_25" at 581,170 size 44x16; Text '工作台'
   Circle "圆_14" at 224,141 size 27x27
      Appearance <- "调整开关"
   TextField "文本域_26" at 217,171 size 44x16; Text '工作台'
   Circle "圆_15" at 535,141 size 27x27
      Appearance <- "工作台顶起压力"
   TextField "文本域_27" at 218,187 size 47x17; Text '进到位'
   TextField "文本域_28" at 265,187 size 33x17; Text '夹紧'
   TextField "文本域_29" at 527,188 size 47x17; Text '夹压力'
   TextField "文本域_30" at 350,171 size 31x16; Text '前左'
   Circle "圆_16" at 352,142 size 27x27
      Appearance <- "工作台落下左前检测"
   TextField "文本域_31" at 345,187 size 47x17; Text '落到位'
   TextField "文本域_32" at 396,171 size 31x16; Text '前右'
   Circle "圆_17" at 396,141 size 27x27
      Appearance <- "工作台落下右前检测"
   TextField "文本域_33" at 391,187 size 47x17; Text '落到位'
   TextField "文本域_34" at 441,170 size 31x16; Text '后左'
   Circle "圆_18" at 442,141 size 27x27
      Appearance <- "工作台落下左后检测"
   TextField "文本域_35" at 437,187 size 47x17; Text '落到位'
   TextField "文本域_36" at 488,170 size 31x16; Text '后右'
   Circle "圆_19" at 488,141 size 27x27
      Appearance <- "工作台落下右边后检测"
   TextField "文本域_37" at 483,188 size 47x17; Text '落到位'
   TextField "文本域_38" at 581,187 size 45x16; Text '夹紧OK'
   TextField "文本域_39" at 304,171 size 44x16; Text '工作台'
   Circle "圆_20" at 311,143 size 27x27
      Appearance <- "工作台落下夹紧(2)"
   TextField "文本域_40" at 302,187 size 47x17; Text '夹紧阀'
   TextField "文本域_20" at 52,232 size 125x27; Text '工作台开进'
   TextField "文本域_41" at 58,306 size 125x27; Text '工作台开出'
   Circle "圆_21" at 227,224 size 27x27
      Appearance <- "上死点"
   TextField "文本域_43" at 220,256 size 44x16; Text '上死点'
   Circle "圆_23" at 276,224 size 27x27
      Appearance <- "调整开关"
   TextField "文本域_46" at 273,257 size 31x16; Text '调整'
   TextField "文本域_47" at 272,274 size 33x17; Text '开关'
   TextField "文本域_50" at 402,255 size 44x16; Text '工作台'
   Circle "圆_25" at 404,224 size 27x27
      Appearance <- "工作台开进"
   TextField "文本域_51" at 397,272 size 35x17; Text '进'
   TextField "文本域_52" at 447,255 size 44x16; Text '工作台'
   Circle "圆_26" at 452,224 size 27x27
      Appearance <- "工作台开进到位"
   TextField "文本域_53" at 444,273 size 47x17; Text '进到位'
   TextField "文本域_59" at 356,256 size 44x16; Text '工台变'
   Circle "圆_29" at 363,224 size 27x27
      Appearance <- "开工作台变频器正常"
   TextField "文本域_60" at 354,272 size 47x17; Text '频正常'
   Circle "圆_12" at 316,224 size 27x27
      Appearance <- "工作台放松OK"
   TextField "文本域_42" at 309,256 size 44x16; Text '工作台'
   TextField "文本域_48" at 309,273 size 45x16; Text '松开OK'
   Circle "圆_22" at 230,305 size 27x27
      Appearance <- "上死点"
   TextField "文本域_44" at 223,337 size 44x16; Text '上死点'
   Circle "圆_24" at 279,305 size 27x27
      Appearance <- "调整开关"
   TextField "文本域_45" at 276,338 size 31x16; Text '调整'
   TextField "文本域_49" at 275,355 size 33x17; Text '开关'
   TextField "文本域_54" at 405,336 size 44x16; Text '工作台'
   Circle "圆_27" at 407,305 size 27x27
      Appearance <- "工作台开出"
   TextField "文本域_55" at 400,353 size 19x17; Text '出'
   TextField "文本域_56" at 450,336 size 44x16; Text '工作台'
   Circle "圆_28" at 455,305 size 27x27
      Appearance <- "工作台顶起右前检测"
   TextField "文本域_57" at 447,354 size 47x17; Text '出到位'
   TextField "文本域_58" at 359,337 size 44x16; Text '工台变'
   Circle "圆_30" at 366,305 size 27x27
      Appearance <- "开工作台变频器正常"
   TextField "文本域_61" at 357,353 size 47x17; Text '频正常'
   Circle "圆_31" at 319,305 size 27x27
      Appearance <- "工作台放松OK"
   TextField "文本域_62" at 312,337 size 44x16; Text '工作台'
   TextField "文本域_63" at 312,354 size 45x16; Text '松开OK'

screen "气垫操作" 800x480
   Button "按钮_1" at 28,424 size 67x56; TextOn '滑块角度'; TextOff '滑块角度'
      on Click: ActivateScreen("滑块角度", 0)
   Button "按钮_2" at 96,424 size 67x56; TextOn '设备状态'; TextOff '设备状态'
      on Click: ActivateScreen("设备状态", 0)
   Button "按钮_3" at 163,424 size 71x55; TextOn '工作台操作'; TextOff '工作台操作'
      on Click: ActivateScreen("工作台操作", 0)
   Button "按钮_4" at 235,424 size 69x56; TextOn '气垫操作'; TextOff '气垫操作'
      on Click: ActivateScreen("气垫操作", 0)
   Button "按钮_5" at 304,423 size 66x57; TextOn '故障显示'; TextOff '故障显示'
      on Click: ActivateScreen("故障显示", 0)
   Button "按钮_6" at 371,423 size 73x57; TextOn '输出显示'; TextOff '输出显示'
      on Click: ActivateScreen("输出显示", 0)
   Button "按钮_7" at 445,422 size 66x58; TextOn '输入显示'; TextOff '输入显示'
      on Click: ActivateScreen("输入显示", 0)
   Button "按钮_8" at 514,423 size 68x56; TextOn '滑块调整'; TextOff '滑块调整'
      on Click: ActivateScreen("滑块调整", 0)
   Button "按钮_9" at 592,422 size 65x58; TextOn '报警信息'; TextOff '报警信息'
      on Click: ActivateScreen("报警信息", 0)
   TextField "文本域_1" at 55,82 size 101x27; Text '气垫上调'
   TextField "文本域_2" at 58,142 size 101x27; Text '气垫下调'
   TextField "文本域_13" at 215,111 size 44x16; Text '上死点'
   TextField "文本域_5" at 304,112 size 70x16; Text '气垫落到位'
   TextField "文本域_3" at 216,176 size 44x16; Text '上死点'
   TextField "文本域_4" at 305,177 size 70x16; Text '气垫落到位'

screen "滑块调整" 800x480
   Button "按钮_1" at 28,424 size 67x56; TextOn '滑块角度'; TextOff '滑块角度'
      on Click: ActivateScreen("滑块角度", 0)
   Button "按钮_2" at 96,424 size 67x56; TextOn '设备状态'; TextOff '设备状态'
      on Click: ActivateScreen("设备状态", 0)
   Button "按钮_3" at 163,424 size 71x55; TextOn '工作台操作'; TextOff '工作台操作'
      on Click: ActivateScreen("工作台操作", 0)
   Button "按钮_4" at 235,424 size 69x56; TextOn '气垫操作'; TextOff '气垫操作'
      on Click: ActivateScreen("气垫操作", 0)
   Button "按钮_5" at 304,423 size 66x57; TextOn '故障显示'; TextOff '故障显示'
      on Click: ActivateScreen("故障显示", 0)
   Button "按钮_6" at 371,423 size 73x57; TextOn '输出显示'; TextOff '输出显示'
      on Click: ActivateScreen("输出显示", 0)
   Button "按钮_7" at 445,422 size 66x58; TextOn '输入显示'; TextOff '输入显示'
      on Click: ActivateScreen("输入显示", 0)
   Button "按钮_8" at 514,423 size 68x56; TextOff '滑块调整'
      on Click: ActivateScreen("滑块调整", 0)
   TextField "文本域_1" at 157,34 size 61x29; Text '1220'
   TextField "文本域_2" at 26,34 size 109x29; Text '滑块上限'
   TextField "文本域_3" at 158,107 size 47x29; Text '560'
   TextField "文本域_4" at 27,107 size 109x29; Text '滑块下限'
   TextField "文本域_6" at 268,33 size 135x29; Text '滑块当前值'
   TextField "文本域_8" at 270,108 size 135x29; Text '滑块设定值'
   Circle "圆_1" at 584,30 size 39x39
      Appearance <- "滑块调整手动/自动"
   Circle "圆_2" at 690,31 size 39x39
      Appearance <- "滑块调整手动/自动"
   TextField "文本域_16" at 583,76 size 41x21; Text '手动'
   TextField "文本域_19" at 689,76 size 41x21; Text '自动'
   IOField "I/O 域_1" at 414,102 size 103x47; FormatPattern 9999
      ProcessValue <- "ECamdata _DB_D{10}滑块设定高度(1)"
   IOField "I/O 域_2" at 414,33 size 103x47; FormatPattern 9999
      ProcessValue <- "ECamdata _DB_D107"
   Switch "开关_1" at 600,93 size 120x56; CaptionText 'Switch'; TextOff '手动'; TextOn '自动'
      on SwitchOff: ResetBit("滑块调整手动/自动")
      on SwitchOn: SetBit("滑块调整手动/自动")
      Appearance <- "滑块调整手动/自动"
      ProcessValue <- "滑块调整手动/自动"
   TextField "文本域_5" at 599,150 size 123x21; Text '手动/自动调整'
   Button "按钮_10" at 592,422 size 65x58; TextOn '报警信息'; TextOff '报警信息'
      on Click: ActivateScreen("报警信息", 0)
   Circle "圆_3" at 32,290 size 33x33
      Appearance <- "平衡缸气压检测"
   TextField "文本域_7" at 8,8 size 37x17; Text 'Text'
   TextField "文本域_10" at 16,300 size 61x17; Text '平衡气压'
   Circle "圆_4" at 97,290 size 33x33
      Appearance <- "液压保护正常指示"
   TextField "文本域_11" at 81,299 size 61x17; Text '液压保护'
   Circle "圆_5" at 156,290 size 33x33
      Appearance <- "润滑正常"
   TextField "文本域_12" at 145,300 size 61x17; Text '润滑正常'
   Circle "圆_6" at 222,290 size 33x33
      Appearance <- "滑块调整电机空开"
   TextField "文本域_13" at 210,301 size 61x17; Text '调整空开'
   Circle "圆_7" at 281,290 size 33x33
      Appearance <- "滑块调整选择开关"
   TextField "文本域_14" at 274,294 size 47x17; Text '滑块调'
   Circle "圆_8" at 335,275 size 33x33
      Appearance <- "上死点"
   TextField "文本域_15" at 326,284 size 47x17; Text '上死点'
   Circle "圆_9" at 439,276 size 33x33
      Appearance <- "滑块调整上极限"
   TextField "文本域_17" at 429,288 size 47x17; Text '上限位'
   Circle "圆_10" at 439,310 size 33x33
      Appearance <- "滑块调整下极限"
   TextField "文本域_18" at 430,319 size 47x17; Text '下限位'
   Circle "圆_11" at 569,275 size 33x33
      Appearance <- "滑块调整向上"
   TextField "文本域_20" at 554,282 size 61x17; Text '调整向上'
   Circle "圆_12" at 570,309 size 33x33
      Appearance <- "滑块调整向下"
   TextField "文本域_21" at 552,318 size 61x17; Text '调整向下'
   Circle "圆_13" at 386,291 size 33x33
      Appearance <- "急停故障(2)"
   TextField "文本域_9" at 385,302 size 33x17; Text '急停'
   Circle "圆_14" at 495,256 size 35x35
      Appearance <- "滑块调整手动/自动"
   TextField "文本域_22" at 494,267 size 41x21; Text '手动'
   Circle "圆_15" at 496,291 size 37x37
      Appearance <- "滑块调整手动/自动"
   TextField "文本域_23" at 491,299 size 41x21; Text '自动'
   Circle "圆_16" at 495,326 size 36x36
      Appearance <- "滑块调整手动/自动"
   TextField "文本域_24" at 494,334 size 41x21; Text '手动'
   TextField "文本域_26" at 275,308 size 47x17; Text '整选择'
   Circle "圆_18" at 334,310 size 33x33
      Appearance <- "下死点"
   TextField "文本域_27" at 325,319 size 47x17; Text '下死点'

screen "报警信息" 800x480
   AlarmView "报警视图_1" at 10,90 size 780x331
   Clock "时钟_1" at 630,64 size 164x20
   GraphicView "图形视图_2" at 2,9 size 78x46; Picture "方鼎LOGO"
   TextField "文本域_5" at 222,19 size 365x33; Text '湖北方鼎科技发展有限公司'
   TextField "文本域_3" at 710,9 size 75x21; Text 'SIEMENS'
   TextField "文本域_4" at 702,37 size 93x17; Text 'SIMATIC HMI'
   TextField "文本域_1" at 325,62 size 109x29; Text '报警信息'
   Button "按钮_1" at 28,424 size 67x56; TextOn '滑块角度'; TextOff '滑块角度'
      on Click: ActivateScreen("滑块角度", 0)
   Button "按钮_2" at 96,424 size 67x56; TextOn '设备状态'; TextOff '设备状态'
      on Click: ActivateScreen("设备状态", 0)
   Button "按钮_3" at 163,424 size 71x55; TextOn '工作台操作'; TextOff '工作台操作'
      on Click: ActivateScreen("工作台操作", 0)
   Button "按钮_4" at 235,424 size 69x56; TextOn '气垫操作'; TextOff '气垫操作'
      on Click: ActivateScreen("气垫操作", 0)
   Button "按钮_5" at 304,423 size 66x57; TextOn '故障显示'; TextOff '故障显示'
      on Click: ActivateScreen("故障显示", 0)
   Button "按钮_6" at 371,423 size 73x57; TextOn '输出显示'; TextOff '输出显示'
      on Click: ActivateScreen("输出显示", 0)
   Button "按钮_7" at 445,422 size 66x58; TextOn '输入显示'; TextOff '输入显示'
      on Click: ActivateScreen("输入显示", 0)
   Button "按钮_8" at 514,423 size 68x56; TextOn '滑块调整'; TextOff '滑块调整'
      on Click: ActivateScreen("滑块调整", 0)
   Button "按钮_9" at 592,422 size 65x58; TextOn '报警信息'; TextOff '报警信息'
      on Click: ActivateScreen("报警信息", 0)

screen "行程控制" 800x480
   Button "按钮_1" at 28,424 size 67x56; TextOn '滑块角度'; TextOff '滑块角度'
      on Click: ActivateScreen("滑块角度", 0)
   Button "按钮_2" at 96,424 size 67x56; TextOn '设备状态'; TextOff '设备状态'
      on Click: ActivateScreen("设备状态", 0)
   Button "按钮_3" at 163,424 size 71x55; TextOn '工作台操作'; TextOff '工作台操作'
      on Click: ActivateScreen("工作台操作", 0)
   Button "按钮_4" at 235,424 size 69x56; TextOn '气垫操作'; TextOff '气垫操作'
      on Click: ActivateScreen("气垫操作", 0)
   Button "按钮_5" at 304,423 size 66x57; TextOn '故障显示'; TextOff '故障显示'
      on Click: ActivateScreen("故障显示", 0)
   Button "按钮_6" at 371,423 size 73x57; TextOn '输出显示'; TextOff '输出显示'
      on Click: ActivateScreen("输出显示", 0)
   Button "按钮_7" at 445,422 size 66x58; TextOn '输入显示'; TextOff '输入显示'
      on Click: ActivateScreen("输入显示", 0)
   Button "按钮_8" at 514,423 size 68x56; TextOn '滑块调整'; TextOff '滑块调整'
      on Click: ActivateScreen("滑块调整", 0)
   Button "按钮_9" at 667,421 size 65x58; TextOn '报警信息'; TextOff '报警信息'
      on Click: ActivateScreen("报警信息", 0)
   Button "按钮_10" at 585,423 size 77x55; TextOn '行程控制'; TextOff '行程控制'
      on Click: ActivateScreen("行程控制", 0)
   Circle "圆_1" at 162,107 size 34x34
      Appearance <- "行程选择"
   TextField "文本域_1" at 153,147 size 61x17; Text '行程选择'
   Circle "圆_2" at 223,107 size 34x34
      Appearance <- "左后双手使用"
   TextField "文本域_2" at 214,147 size 61x17; Text '左前选择'
   Circle "圆_3" at 284,107 size 34x34
      Appearance <- "右前双手选择"
   TextField "文本域_3" at 275,147 size 61x17; Text '右前选择'
   Circle "圆_4" at 345,107 size 34x34
      Appearance <- "行程选择"
   TextField "文本域_4" at 336,147 size 61x17; Text '换模完成'
   Circle "圆_5" at 406,107 size 34x34
      Appearance <- "行程选择"
   TextField "文本域_5" at 397,147 size 61x17; Text '急停正常'
   Circle "圆_6" at 467,107 size 34x34
      Appearance <- "行程选择"
   TextField "文本域_6" at 453,163 size 75x17; Text '主电机运行'
   Circle "圆_7" at 528,107 size 34x34
      Appearance <- "行程选择"
   TextField "文本域_7" at 519,147 size 61x17; Text '设备正常'
   Circle "圆_8" at 589,107 size 34x34
      Appearance <- "行程选择"
   TextField "文本域_8" at 580,147 size 61x17; Text '润滑正常'
   Button "按钮_11" at 0,3 size 165x55; TextOn '行程控制'; TextOff '行程控制'
      on Click: ActivateScreen("行程控制", 0)
   TextField "文本域_20" at 318,71 size 125x27; Text '主电机启动'

screen "主电机启动" 800x480
   TextField "文本域_20" at 111,181 size 125x27; Text '主电机启动'
   Circle "圆_21" at 286,176 size 33x33
      Appearance <- "润滑正常"
   TextField "文本域_43" at 279,231 size 57x16; Text '润滑正常'
   Circle "圆_23" at 346,176 size 33x33
      Appearance <- "调整开关"
   TextField "文本域_46" at 343,232 size 44x16; Text '润滑正'
   TextField "文本域_47" at 342,249 size 47x17; Text '常指示'
   TextField "文本域_50" at 523,230 size 57x16; Text '启动延时'
   Circle "圆_25" at 525,175 size 35x35
      Appearance <- "工作台开进"
   TextField "文本域_52" at 584,230 size 70x16; Text '主电机运行'
   Circle "圆_26" at 589,175 size 35x35
      Appearance <- "工作台开进到位"
   TextField "文本域_59" at 456,231 size 57x16; Text '变频上电'
   Circle "圆_29" at 463,176 size 34x34
      Appearance <- "开工作台变频器正常"
   Circle "圆_12" at 404,176 size 33x33
      Appearance <- "工作台放松OK"
   TextField "文本域_42" at 395,231 size 57x16; Text '正转条件'
   TextField "文本域_48" at 397,248 size 12x16; Text 'Text'
   IOField "I/O 域_1" at 0,0 size 96x32; FormatPattern 1
      ProcessValue <- "润滑电机工作指示"
   IOField "I/O 域_2" at 0,0 size 96x32; FormatPattern 1
      ProcessValue <- "润滑电机工作指示"
   IOField "I/O 域_3" at 0,0 size 96x32; FormatPattern 1
      ProcessValue <- "润滑电机工作指示"
   IOField "I/O 域_4" at 0,0 size 96x32; FormatPattern 1
      ProcessValue <- "正转条件"
   IOField "I/O 域_5" at 0,0 size 96x32; FormatPattern 1
      ProcessValue <- "主电机启动指示"
*)